PROGRAM MAIN
VAR
	counterOne : DINT;
END_VAR

counterOne := counterOne + 1;
IF counterOne > 20000 THEN
	counterOne := 0;
END_IF

END_PROGRAM

(* stored: Version 1.1.0.1, ProductVersion 3.1.4024.12
   POU MAIN: Id {7a46fe8f-c07c-4967-a6f0-adc22ff4f012}, SpecialFunc None *)
